Staubli VAL3: RefreshList.pgx

program RefreshList()
  local num l_ni
begin
  //
  if bListRefresh
    switch nPage
      case 0
        resize(sList,1,2)
        for l_ni=0 to 1
          sList[l_ni]="pallet"+toString("",l_ni+1)
        endFor
      break

      case 1

      break
    endSwitch
  endIf

end
